// TIA Portal V19 export
DATA_BLOCK "DI_FW_1"   // DB11
AUTHOR : MS
VERSION : 0.0
// stored: AutoNumber false, InstanceOfName FB_FW_x, InstanceOfType FB
"FB_FW_x"
   // VAR RETAIN
   //    ZST : Struct
   //       BEREIT : Bool := TRUE;
   //       AKTIV : Bool := FALSE;
   //       FEHLER : Bool := FALSE;
   //       REFERENZIERT : Bool := TRUE;
   //       HEBEN_AKT : Bool := FALSE;
   //       SENKEN_AKT : Bool := FALSE;
   //       VORWAERTS_AKT : Bool := FALSE;
   //       RUECKWAERTS_AKT : Bool := FALSE;
   //       Befehl_ok : Bool := FALSE;
   //       Befehl_nok : Bool := FALSE;
   //       Befehl_done : Bool := TRUE;
   //       Tipp : Bool := FALSE;
   //       Hand : Bool := TRUE;
   //       Auto_Stop : Bool := FALSE;
   //       Auto : Bool := FALSE;
   //       Semi : Bool := FALSE;
   //       POSITION_li : Byte := 16#05;
   //       Ebene_li : Byte := 16#01;
   //       PosInc : DInt := 4748;
   //       HubInc_li : DInt := 403;
   //       Oben_li : Bool := FALSE;
   //       Z_Sensor_li : Bool := FALSE;
   //       Unten_li : Bool := TRUE;
   //       HubSensor_li : Bool := TRUE;
   //       low_SU_li : Bool := FALSE;
   //       Mittig : Bool := FALSE;
   //       HW_mittig : Bool := FALSE;
   //       old_vor : Bool := TRUE;
   //       schieben : Bool := FALSE;
   //       SoftStop : Bool := FALSE;
   //       Halt : Bool := FALSE;
   //       Ofs_mittig : Bool := TRUE;
   //       PosStop : Bool := TRUE;
   //       schieben_erlaubt : Bool := FALSE;
   //       Ofs_Bereich : Bool := FALSE;
   //       free : Bool := FALSE;
   //       POSITION_re : Byte := 16#06;
   //       Ebene_re : Byte := 16#01;
   //       Oben_re : Bool := FALSE;
   //       Z_Sensor_re : Bool := FALSE;
   //       Unten_re : Bool := TRUE;
   //       HubSensor_re : Bool := TRUE;
   //       low_SU_re : Bool := FALSE;
   //       res165 : Bool := FALSE;
   //       res166 : Bool := FALSE;
   //       res167 : Bool := FALSE;
   //       Res_B17 : Byte := 16#00;
   //       WT_DB_NR_li : Byte := 16#00;
   //       WT_DB_NR_re : Byte := 16#00;
   //       WT_NR_LANG_li : DWord := 16#0000_0000;
   //       Befehl_akt : Byte := 16#00;
   //       UP_ON : Bool := FALSE;
   //       next_Step : Bool := FALSE;
   //       new_Bef : Bool := TRUE;
   //       MicM1 : Bool := FALSE;
   //       MicM2 : Bool := FALSE;
   //       MicM3 : Bool := FALSE;
   //       MicM4 : Bool := FALSE;
   //       Start_UP : Bool := FALSE;
   //       Adr_Next_Step : Word := 16#0000;
   //       UP_RET_ADR : Word := 16#0000;
   //       BEFEHL : DWord := 16#0000_0000;
   //       Verweil : DInt := 0;
   //       SchiebeInc : DInt := 0;
   //       Speed_Fahrt : Int := 0;
   //       Speed_Hub_li : Int := 0;
   //       Rest_Zeit : DInt := 0;
   //    END_STRUCT;
   //    IN : Struct
   //       DIR_VOR : Bool := FALSE;
   //       DIR_RCK : Bool := FALSE;
   //       Anf_Hub_li : Bool := FALSE;
   //       Anf_Hub_re : Bool := FALSE;
   //       DIR_HEB_li : Bool := FALSE;
   //       DIR_SENK_li : Bool := FALSE;
   //       DIR_HEB_re : Bool := FALSE;
   //       DIR_SENK_re : Bool := FALSE;
   //       Knauf_Auto : Bool := FALSE;
   //       Aktion : Bool := TRUE;
   //       Halt : Bool := FALSE;
   //       REP_TASTE : Bool := FALSE;
   //       QUITT_ALARM : Bool := FALSE;
   //       Unten : Bool := TRUE;
   //       Oben : Bool := FALSE;
   //       Laser_on : Bool := TRUE;
   //       BA_Tipp_ext : Bool := FALSE;
   //       BA_Hand_ext : Bool := TRUE;
   //       BA_Auto_Stop_ext : Bool := FALSE;
   //       BA_Auto_ext : Bool := FALSE;
   //       Unten_li : Bool := FALSE;
   //       Oben_li : Bool := FALSE;
   //       Unten_re : Bool := FALSE;
   //       Oben_re : Bool := FALSE;
   //       FahrBreak_on : Bool := FALSE;
   //       HubBreak_on : Bool := FALSE;
   //       Pos_ok : Bool := TRUE;
   //       Hub_ok_li : Bool := TRUE;
   //       Com_Reset : Bool := FALSE;
   //       Hub_ok_re : Bool := TRUE;
   //       PosGr_min : Bool := TRUE;
   //       PosGr_max : Bool := TRUE;
   //       Grenze_min : DInt := 740;
   //       Grenze_max : DInt := 29010;
   //    END_STRUCT;
   //    ErrIn : Struct
   //       Alarm : Struct
   //          NotHalt : Bool := FALSE;
   //          PosSys : Bool := FALSE;
   //          HubSys_li : Bool := FALSE;
   //          HubSys_re : Bool := FALSE;
   //          Hub_nok_links : Bool := FALSE;
   //          Hub_nok_rechts : Bool := FALSE;
   //          Fahrt_nok : Bool := FALSE;
   //          POS_BELEGT_li : Bool := FALSE;
   //          POS_BELEGT_re : Bool := FALSE;
   //          BE_Vor : Bool := FALSE;
   //          BE_Rck : Bool := FALSE;
   //          Koll_LF : Bool := FALSE;
   //          Koll_WF : Bool := FALSE;
   //          AFS_BS : Bool := FALSE;
   //          AFS_WS : Bool := FALSE;
   //          Gurt_UP_links : Bool := FALSE;
   //          Gurt_DN_links : Bool := FALSE;
   //          Gurt_UP_rechts : Bool := FALSE;
   //          Gurt_DN_rechts : Bool := FALSE;
   //          Last_UeW_links : Bool := FALSE;
   //          Last_UeW_rechts : Bool := FALSE;
   //          F_Brk_Hub_links : Bool := FALSE;
   //          F_Brk_Hub_rechts : Bool := FALSE;
   //          F_Brk_Fahr : Bool := FALSE;
   //          Gurt_UeL_links : Bool := FALSE;
   //          Gurt_UeL_rechts : Bool := FALSE;
   //          Profinet_IO_nok : Bool := FALSE;
   //          Al_res_8 : Bool := FALSE;
   //          AL_res_9 : Bool := FALSE;
   //          AL_res_10 : Bool := FALSE;
   //          AL_res_11 : Bool := FALSE;
   //          AL_res_12 : Bool := FALSE;
   //       END_STRUCT;
   //       Warnung : Struct
   //          Wrn_Optik_PosSys : Bool := FALSE;
   //          Wrn_Temp_PosSys : Bool := FALSE;
   //          Wrn_Plaus_PosSys : Bool := FALSE;
   //          Wrn_WZ_niO_li_1 : Bool := FALSE;
   //          Wrn_WZ_niO_li_2 : Bool := FALSE;
   //          Wrn_WZ_niO_li_3 : Bool := FALSE;
   //          Wrn_WZ_niO_li_4 : Bool := FALSE;
   //          Wrn_WZ_niO_re_1 : Bool := FALSE;
   //          Wrn_WZ_niO_re_2 : Bool := FALSE;
   //          Wrn_WZ_niO_re_3 : Bool := FALSE;
   //          Wrn_WZ_niO_re_4 : Bool := FALSE;
   //          Wrn_res_10 : Bool := FALSE;
   //          Wrn_res_11 : Bool := FALSE;
   //          Wrn_WT_nUmsetzbar : Bool := FALSE;
   //          Wrn_Temp_Fahr : Bool := FALSE;
   //          Wrn_Temp_Hub : Bool := FALSE;
   //       END_STRUCT;
   //    END_STRUCT;
   //    OUT : Struct
   //       VOR : Bool := FALSE;
   //       RUECK : Bool := FALSE;
   //       POS_EIL : Bool := FALSE;
   //       HEBEN : Bool := FALSE;
   //       SENKEN : Bool := FALSE;
   //       HUB_EIL_li : Bool := FALSE;
   //       HUB_EIL_re : Bool := FALSE;
   //       HEBEN_li : Bool := FALSE;
   //       HEBEN_re : Bool := FALSE;
   //       SENKEN_li : Bool := FALSE;
   //       SENKEN_re : Bool := FALSE;
   //       res_3 : Bool := FALSE;
   //       res_4 : Bool := FALSE;
   //       res_5 : Bool := FALSE;
   //       res_6 : Bool := FALSE;
   //       res_7 : Bool := FALSE;
   //       res_8 : Bool := FALSE;
   //       res_9 : Bool := FALSE;
   //       TIPP : Bool := FALSE;
   //       Req_Laser : Bool := TRUE;
   //       no_Brms : Bool := FALSE;
   //       res_12 : Bool := FALSE;
   //       res_13 : Bool := FALSE;
   //       res_14 : Bool := FALSE;
   //       res_15 : Bool := FALSE;
   //       res_16 : Bool := FALSE;
   //       res_17 : Bool := FALSE;
   //       res_18 : Bool := FALSE;
   //       res_19 : Bool := FALSE;
   //       res_20 : Bool := FALSE;
   //       res_21 : Bool := FALSE;
   //       Parken : Bool := FALSE;
   //    END_STRUCT;
   //    Micro : Struct
   //       Adr_UP : Array[1..15] of Word;
   //       Liste : Array[0..79] of Byte;
   //    END_STRUCT;
   //    PAR : Struct
   //       FW_Nr : Byte := 16#01;
   //       Wichtung : Byte := 16#00;
   //       TIMER_NR : Int := 10;
   //       Reihe : Byte := 16#01;
   //       resB : Byte := 16#00;
   //       Vorzugsbereich_min : Byte := 16#00;
   //       Vorzugsbereich_max : Byte := 16#00;
   //       Aktionsbereich_min : Byte := 16#00;
   //       Aktionsbereich_max : Byte := 16#00;
   //       resInt : Int := 0;
   //       Fahrt : Struct
   //          FAHRBEREICH_MIN : Byte := 16#01;
   //          FAHRBEREICH_MAX : Byte := 16#1F;
   //          REF_Pos : Byte := 16#00;
   //          Abstand_vor : DInt := 2000;
   //          dyn_Eil : DInt := 0;
   //          MessOffset : DInt := 0;
   //          Dir_negativ : Byte := 16#00;
   //          ErrCount : Byte := 16#14;
   //          Bereich_Pos : DInt := 10;
   //          resD : DInt := 0;
   //          Bereich_Ziel : DInt := 5;
   //          max_Anhalteweg : DInt := 170;
   //          Bereich_lngsm : DInt := 0;
   //          TO_Fahren : S5Time := S5T#5S;
   //          Offset_SoftStop : Int := 0;
   //          delta_s : Int := 10;
   //          resT : S5Time := S5T#0MS;
   //          WT_Speed : Int := 100;
   //          Park_Pos : Int := 0;
   //          Count_Park : Int := 0;
   //          Fahr_DBNr : Int := 21;
   //       END_STRUCT;
   //       Hub : Struct
   //          Hub_DBNr : Int := 22;
   //          WT_Speed : Int := 100;
   //          resInt : Int := 0;
   //          Dir_negativ_re : Byte := 16#01;
   //          ErrCount_re : Byte := 16#14;
   //          MessOffset_li : DInt := 1000;
   //          Dir_negativ_li : Byte := 16#01;
   //          ErrCount_li : Byte := 16#14;
   //          Bereich_Pos : DInt := 10;
   //          resD : DInt := 0;
   //          Bereich_Ziel : DInt := 5;
   //          MessOffset_re : DInt := 1000;
   //          Bereich_lngsm : DInt := 0;
   //          TO_Heben_Senken_hi : S5Time := S5T#10S;
   //          TO_Heben_Senken_low : S5Time := S5T#20S;
   //          delta_s : Int := 1;
   //          TO_HW : S5Time := S5T#10S;
   //          TV_HubSensor : S5Time := S5T#0MS;
   //          Ebene0 : DInt := 100;
   //          Ebene1 : DInt := 400;
   //          Ebene2 : DInt := 1600;
   //          Ebene3 : DInt := 2400;
   //          Ebene4 : DInt := 0;
   //          Ebene5 : DInt := 0;
   //          Ebene6 : DInt := 0;
   //          Ebene7 : DInt := 0;
   //          SU_Ebenen : Byte := 16#07;
   //          Z_Ebene : Byte := 16#00;
   //          SO_Ebene : Byte := 16#03;
   //          SUF_Ebene : Byte := 16#01;
   //       END_STRUCT;
   //       Free : Struct
   //          TDR_Pause : Int := 0;
   //          TDR_Drehen : Int := 0;
   //          Ziel_Inc : DWord := 16#0000_0000;
   //          resW3 : Word := 16#0000;
   //          TS_Ablasszeit : Int := 0;
   //          TS_MV_Zeit : Int := 0;
   //          TS_Takte_leeren : Byte := 16#00;
   //          TS : Bool := FALSE;
   //          FG_Leeren : Bool := FALSE;
   //          TS_Ablass_Sonderpos : Bool := FALSE;
   //          res153 : Bool := FALSE;
   //          res154 : Bool := FALSE;
   //          res155 : Bool := FALSE;
   //          Z_no_Brms : Bool := FALSE;
   //          Laser_req : Bool := TRUE;
   //          Laser : DWord := 16#0000_0000;
   //       END_STRUCT;
   //    END_STRUCT;
   //    TMP : Struct
   //       Hub_Ebenen : Byte := 16#0B;
   //       Zielebene_re : Byte := 16#00;
   //       Zielebene_li : Byte := 16#00;
   //       ZielPos : Byte := 16#00;
   //       HubZielInc_li : DInt := 0;
   //       FahrZielInc : DInt := 0;
   //       low_SU_Ebene : Byte := 16#00;
   //       ErrCount_Possys : Byte := 16#00;
   //       FHLR_NR : Int := 97;
   //       CouPHub : Int := 0;
   //       EndZiel : Int := 0;
   //       count1 : Int := 0;
   //       count2 : Int := 0;
   //       count3 : Int := 0;
   //       count4 : Int := 0;
   //       count5 : Int := 0;
   //       Verweil : DInt := 0;
   //       Dauer : DInt := 0;
   //       SoftStopInc : DInt := 29000;
   //       Opt_Start_Pos : Byte := 16#00;
   //       Opt_Ziel_Pos : Byte := 16#00;
   //       Zustand : Byte := 16#00;
   //       Count_TS_leeren : Byte := 16#00;
   //       HW_akt_li : Bool := FALSE;
   //       HW_akt_re : Bool := FALSE;
   //       FM_F_Taste : Bool := FALSE;
   //       res : Bool := TRUE;
   //       DKL_Sperre : Bool := FALSE;
   //       FM_low_SU_li : Bool := FALSE;
   //       FW_gestartet : Bool := FALSE;
   //       old_hub : Bool := FALSE;
   //       old_vor_hoch : Bool := FALSE;
   //       old_rueck_runter : Bool := FALSE;
   //       FM_low_SU_re : Bool := FALSE;
   //       FP_K_Auto : Bool := FALSE;
   //       FP_K_Auto_int : Bool := FALSE;
   //       noATZ : Bool := FALSE;
   //       noPend : Bool := FALSE;
   //       nextQ_Takt : Bool := FALSE;
   //       nexQuelle : Word := 16#0000;
   //       AltPos : DInt := 4740;
   //       AltHub_li : DInt := 403;
   //    END_STRUCT;
   //    MLD : Struct
   //       Alarm_HW : Struct
   //          PosSys : Bool := FALSE;
   //          BE_rck : Bool := FALSE;
   //          BE_vor : Bool := FALSE;
   //          HubSys_li : Bool := FALSE;
   //          HubSys_re : Bool := FALSE;
   //          GE_oben_li : Bool := FALSE;
   //          GE_unten_li : Bool := FALSE;
   //          GE_oben_re : Bool := FALSE;
   //          GE_unten_re : Bool := FALSE;
   //          Koll_LF : Bool := FALSE;
   //          Koll_WF : Bool := FALSE;
   //          Afs_BS : Bool := FALSE;
   //          Afs_WS : Bool := FALSE;
   //          GurtUeL_li : Bool := FALSE;
   //          GurtUeL_re : Bool := FALSE;
   //          St_FU_Fahrt : Bool := FALSE;
   //          F_Brk_Hub_li : Bool := FALSE;
   //          F_Brk_Hub_re : Bool := FALSE;
   //          F_Brk_Fahr : Bool := FALSE;
   //          St_FU_Hub_li : Bool := FALSE;
   //          St_FU_Hub_re : Bool := FALSE;
   //          Last_UeW_li : Bool := FALSE;
   //          Last_UeW_re : Bool := FALSE;
   //          Temp_Fahrt : Bool := FALSE;
   //          Temp_Hub : Bool := FALSE;
   //          Laser_TF : Bool := FALSE;
   //          Laser_PL : Bool := FALSE;
   //          Profinet_nok : Bool := FALSE;
   //          res_1 : Bool := FALSE;
   //          res_2 : Bool := FALSE;
   //          res_3 : Bool := FALSE;
   //          res_4 : Bool := FALSE;
   //       END_STRUCT;
   //       Alarm_SW : Struct
   //          Fehler_Quitt : Bool := FALSE;
   //          BA_ungueltig : Bool := FALSE;
   //          ProgErr : Bool := FALSE;
   //          nReferenz : Bool := FALSE;
   //          NotStop : Bool := FALSE;
   //          Laser_off : Bool := FALSE;
   //          TO_Fahrt : Bool := FALSE;
   //          Auto_SU : Bool := FALSE;
   //          Auto_WT : Bool := FALSE;
   //          WT_change : Bool := FALSE;
   //          Hub_not_mittig_li : Bool := FALSE;
   //          Hub_nen_li : Bool := FALSE;
   //          TO_Hub_li : Bool := FALSE;
   //          Senken_WT_li : Bool := FALSE;
   //          Senken_Sperre_li : Bool := FALSE;
   //          Heben_WT_li : Bool := FALSE;
   //          SO_fehlt_li : Bool := FALSE;
   //          SU_fehlt_li : Bool := FALSE;
   //          PosTyp_WT_Typ_li : Bool := FALSE;
   //          WTon_bei_SU_li : Bool := FALSE;
   //          TO_Hub_re : Bool := FALSE;
   //          Senken_WT_re : Bool := FALSE;
   //          Senken_Sperre_re : Bool := FALSE;
   //          Heben_WT_re : Bool := FALSE;
   //          SO_fehlt_re : Bool := FALSE;
   //          SU_fehlt_re : Bool := FALSE;
   //          PosTyp_WT_Typ_re : Bool := FALSE;
   //          WTon_bei_SU_re : Bool := FALSE;
   //          Hub_not_mittig_re : Bool := FALSE;
   //          Hub_nen_re : Bool := FALSE;
   //          ALSW_31 : Bool := FALSE;
   //          TO_Befehl : Bool := FALSE;
   //       END_STRUCT;
   //       Warnung : Struct
   //          Optik_PosSys : Bool := FALSE;
   //          Temp_PosSys : Bool := FALSE;
   //          Temp_Fahrt : Bool := FALSE;
   //          Temp_Hub : Bool := FALSE;
   //          LSA : Bool := FALSE;
   //          Bh0 : Bool := FALSE;
   //          Bh100 : Bool := FALSE;
   //          Bh1000 : Bool := FALSE;
   //          Wrn_Plaus_PosSys : Bool := FALSE;
   //          Wrn_WZ_niO_li_1 : Bool := FALSE;
   //          Wrn_WZ_niO_li_2 : Bool := FALSE;
   //          Wrn_WZ_niO_li_3 : Bool := FALSE;
   //          Wrn_WZ_niO_li_4 : Bool := FALSE;
   //          Wrn_WZ_niO_re_1 : Bool := FALSE;
   //          Wrn_WZ_niO_re_2 : Bool := FALSE;
   //          Wrn_WZ_niO_re_3 : Bool := FALSE;
   //          Wrn_WZ_niO_re_4 : Bool := FALSE;
   //          WARN_18 : Bool := FALSE;
   //          WARN_19 : Bool := FALSE;
   //          WARN_20 : Bool := FALSE;
   //          WARN_21 : Bool := FALSE;
   //          WARN_22 : Bool := FALSE;
   //          WARN_23 : Bool := FALSE;
   //          WARN_24 : Bool := FALSE;
   //          WARN_25 : Bool := FALSE;
   //          WARN_26 : Bool := FALSE;
   //          WARN_27 : Bool := FALSE;
   //          WARN_28 : Bool := FALSE;
   //          WARN_29 : Bool := FALSE;
   //          WARN_30 : Bool := FALSE;
   //          WARN_WT_nUms : Bool := FALSE;
   //          WARN_nAuto : Bool := FALSE;
   //       END_STRUCT;
   //       AM_ALHW : DWord := 16#0000_0000;
   //       AM_ALSW : DWord := 16#0000_0000;
   //       AM_WARN : DWord := 16#0000_0000;
   //    END_STRUCT;
   //    HELP : Struct
   //       Count_PosSys : Int := 0;
   //       Count_Laser_on : Int := 0;
   //       Count_Parkpos : Int := 0;
   //       Endziel_WT : Byte := 16#00;
   //       QTZiel : Byte := 16#00;
   //       Grenze_min : Int := 1;
   //       Grenze_max : Int := 29;
   //       Speed_Hub_re : Int := 0;
   //       ResI_8 : Int := 0;
   //       ResI_9 : Int := 0;
   //       ResI_10 : Int := 0;
   //       AuftragWT_li : DInt := 0;
   //       AuftragWT_re : DInt := 0;
   //       HubInc_re : DInt := 403;
   //       WT_NR_LANG_re : DWord := 16#0000_0000;
   //       HubZielInc_re : DInt := 0;
   //       AltHub_re : DInt := 403;
   //       ResDI_5 : DInt := 0;
   //       ResDI_6 : DInt := 0;
   //       ResDI_7 : DInt := 0;
   //       ResDI_8 : DInt := 0;
   //       Last_1 : Real := 0.0;
   //       Last_2 : Real := 0.0;
   //       WZ_links_1 : Real := 0.0;
   //       WZ_links_2 : Real := 0.0;
   //       WZ_links_3 : Real := 0.0;
   //       WZ_links_4 : Real := 0.0;
   //       WZ_rechts_1 : Real := 0.0;
   //       WZ_rechts_2 : Real := 0.0;
   //       WZ_rechts_3 : Real := 0.0;
   //       WZ_rechts_4 : Real := 0.0;
   //       F_Halt : Bool := FALSE;
   //       T_Halt : Bool := FALSE;
   //       FP_Auto : Bool := FALSE;
   //       res_4 : Bool := FALSE;
   //       res_5 : Bool := FALSE;
   //       res_6 : Bool := FALSE;
   //       res_7 : Bool := FALSE;
   //       res_8 : Bool := FALSE;
   //       res_9 : Bool := FALSE;
   //       res_10 : Bool := FALSE;
   //       res_11 : Bool := FALSE;
   //       res_12 : Bool := FALSE;
   //       res_13 : Bool := FALSE;
   //       res_14 : Bool := FALSE;
   //       res_15 : Bool := FALSE;
   //       res_16 : Bool := FALSE;
   //       res_17 : Bool := FALSE;
   //       res_18 : Bool := FALSE;
   //       res_19 : Bool := FALSE;
   //       res_20 : Bool := FALSE;
   //       res_21 : Bool := FALSE;
   //       res_22 : Bool := FALSE;
   //       res_23 : Bool := FALSE;
   //       res_24 : Bool := FALSE;
   //       res_25 : Bool := FALSE;
   //       res_26 : Bool := FALSE;
   //       res_27 : Bool := FALSE;
   //       res_28 : Bool := FALSE;
   //       res_29 : Bool := FALSE;
   //       res_30 : Bool := FALSE;
   //       Last_button_rck : Bool := FALSE;
   //       Last_button_vor : Bool := TRUE;
   //       Tol_UeW_WZ : Real := 0.0;
   //       AW_WZ_li_vorn : Real := 0.0;
   //       Sum_WZ_li_vorn : Real := 0.0;
   //       AW_WZ_li_hinten : Real := 0.0;
   //       Sum_WZ_li_hinten : Real := 0.0;
   //       AW_WZ_re_vorn : Real := 0.0;
   //       Sum_WZ_re_vorn : Real := 0.0;
   //       AW_WZ_re_hinten : Real := 0.0;
   //       Sum_WZ_re_hinten : Real := 0.0;
   //       Summe_WZ_li : Real := 0.0;
   //       AW_Summe_WZ_li : Real := 0.0;
   //       Summe_WZ_re : Real;
   //       AW_Summe_WZ_re : Real;
   //    END_STRUCT;
   // END_VAR
BEGIN
   Micro.Adr_UP[1] := 16#0066;
   Micro.Adr_UP[2] := 16#006A;
   Micro.Adr_UP[3] := 16#006E;
   Micro.Adr_UP[4] := 16#0077;
   Micro.Adr_UP[5] := 16#007D;
   Micro.Adr_UP[6..13] := 16#0086;
   Micro.Adr_UP[14] := 16#0082;
   Micro.Adr_UP[15] := 16#0084;
   Micro.Liste[0] := 16#02;
   Micro.Liste[1] := 16#14;
   Micro.Liste[2] := 16#05;
   Micro.Liste[3] := 16#00;
   Micro.Liste[4] := 16#03;
   Micro.Liste[5] := 16#14;
   Micro.Liste[6] := 16#05;
   Micro.Liste[7] := 16#00;
   Micro.Liste[8] := 16#01;
   Micro.Liste[9] := 16#15;
   Micro.Liste[10] := 16#04;
   Micro.Liste[11] := 16#0E;
   Micro.Liste[12] := 16#18;
   Micro.Liste[13] := 16#16;
   Micro.Liste[14] := 16#0B;
   Micro.Liste[15] := 16#19;
   Micro.Liste[16] := 16#00;
   Micro.Liste[17] := 16#09;
   Micro.Liste[18] := 16#10;
   Micro.Liste[19] := 16#03;
   Micro.Liste[20] := 16#07;
   Micro.Liste[21] := 16#0C;
   Micro.Liste[22] := 16#00;
   Micro.Liste[23] := 16#14;
   Micro.Liste[24] := 16#09;
   Micro.Liste[25] := 16#11;
   Micro.Liste[26] := 16#12;
   Micro.Liste[27] := 16#00;
   Micro.Liste[28] := 16#0A;
   Micro.Liste[29] := 16#00;
   Micro.Liste[30] := 16#06;
   Micro.Liste[31..79] := 16#00;
END_DATA_BLOCK
